Staubli VAL3: remSetHeartbeat.pgx

program remSetHeartbeat(string& sArgs[] (dimensions=1), string& sReturn[] (dimensions=1))
begin
  // Set the PPS status in the robot
  //
  logMsg("call remSetHeatbeat")
  call remSetnGlobal(sArgs,nHeartbeat,0,5000,"NOTHEARTBEAT",sReturn)
end
